FUNCTION_BLOCK FB_MapStim300
VAR_INPUT
	stFilterParams : ST_FTR_IIRSpec := (
		eFilterName   := E_FTR_Name.eButterworth,
		eFilterType   := E_FTR_Type.eLowPass,
		nFilterOrder  := 2,
		fSamplingRate := 0.001,
		fCutoff       := 4.0,
		nOversamples  := 1,
		nChannels     := 1,
		pInitialValues := ADR(fRollDeg),
		nInitialValuesSize := SIZEOF(fRollDeg)
	);
	
	fbFilter : FB_FTR_IIRSpec := (stConfig := stFilterParams);
END_VAR
VAR_OUTPUT
	ImuData : ST_IMUData;
	
	fRollDegFiltered : LREAL;
	fRollDeg : LREAL;
	fPitchDeg : LREAL;
END_VAR

VAR
		

	//serial communication with el6022
	fbGetSerialData : FB_GetSerialData;	
	ImuRawDataFrame : tDataFrame;
	
	fbEL6022Ctrl       : SerialLineControl;
	bEL6022CtrlError   : BOOL;
   	eEL6022CtrlErrorID : ComError_t;
   
	(* I/O variables for a EL6022 terminal*)
	stIn_EL6022 AT %I*    : EL6inData22B; 		(* linked to the EL6022 in the TwinCAT System Manager *)
	stOut_EL6022 AT %Q*    : EL6outData22B;		(* linked to the EL6022 in the TwinCAT System Manager *)
	
	RxBufferEL : ComBuffer; (* Receive data buffer; used with all receive function blocks *)
	TxBufferEL : ComBuffer; (* Transmit data buffer; used with all receive function blocks *)

	

	fbTimer : TON := (PT := T#1S);
	nCounter : DINT;
	fSampleRate : LREAL;
	
	//COmplementary filter
	fbAccelerometer : FB_AccelerometerAngle;
	fbComplementaryFilterRoll : FB_ComplementaryFilter := (fFilterRatio:=0.98);
	fbComplementaryFilterPitch : FB_ComplementaryFilter := (fFilterRatio:=0.98);
	
	// Task cycle time monitoring
	bFirstRun : BOOL := TRUE;
	Ts : LREAL := 0.01;
	fbGetCurrentTaskIdx : GETCURTASKINDEX;
	bCycleTimeExceeded : BOOL;
	nCycleCount : UDINT;
	
END_VAR

VAR CONSTANT
	header : BYTE := 16#AF;
	nDataSize : UDINT := SIZEOF(tDataFrame);
	fRatioGyro : LREAL := 1.0/EXPT(2,14);
	fRatioAcc : LREAL := 1.0/EXPT(2,19);
END_VAR

IF bFirstRun THEN
	getSampleTIme();
	bFirstRun:= FALSE;
END_IF

fbEL6022Ctrl(
   Mode:= SERIALLINEMODE_EL6_22B, 
   pComIn:= ADR(stIn_EL6022), 
   pComOut:= ADR(stOut_EL6022), 
   SizeComIn:= SIZEOF(stIn_EL6022), 
   Error=> bEL6022CtrlError, 
   ErrorID=> eEL6022CtrlErrorID, 
   TxBuffer:= TxBufferEL, 
   RxBuffer:= RxBufferEL
);

nCounter := nCounter + 1;
fbTimer(IN := TRUE);
IF fbTimer.Q THEN
	fbTimer(IN := FALSE);
	fSampleRate := 1.0/TO_LREAL(nCounter);
	nCounter := 0;
END_IF

fbGetSerialData(
	pHeader := ADR(header),
	cbHeaderSize := 1,
	cbPacketSize := nDataSize,
	stRxBuffer := RxBufferEL,
	pDataBuffer := ADR(ImuRawDataFrame),
	cbDataBufferSize := nDataSize
);

IF fbGetSerialData.NewData THEN
	mapStim300(
		in := ADR(ImuRawDataFrame),
		out := ImuData
	);
	
	fbAccelerometer(fAx:=ImuData.stAcc.x,fAy:=ImuData.stAcc.y,fAz:=ImuData.stAcc.z);
	
	
END_IF

fbComplementaryFilterRoll(fAccAngle:=fbAccelerometer.fRoll,fGyroRate:=ImuData.stGyro.x*CONSTANTS.DEG_TO_RAD,fStepTime:=Ts,fAngle=>ImuData.fRoll);
fbComplementaryFilterPitch(fAccAngle:=fbAccelerometer.fPitch,fGyroRate:=ImuData.stGyro.y*CONSTANTS.DEG_TO_RAD,fStepTime:=Ts,fAngle=>ImuData.fPitch);

fRollDeg := ImuData.fRoll * CONSTANTS.RAD_TO_DEG;
fbFilter.Call(
	pIn := ADR(fRollDeg),
	nSizeIn := SIZEOF(fRollDeg),
	pOut := ADR(fRollDegFiltered),
	nSizeOut := SIZEOF(fRollDegFiltered)
);

fPitchDeg := ImuData.fPitch * CONSTANTS.RAD_TO_DEG;

ACTION getSampleTIme:
// Get sample time of current task
fbGetCurrentTaskIdx();
bCycleTimeExceeded := _TaskInfo[fbGetCurrentTaskIdx.index].CycleTimeExceeded;
nCycleCount := _TaskInfo[fbGetCurrentTaskIdx.index].CycleCount;
Ts := UDINT_TO_LREAL(_TaskInfo[fbGetCurrentTaskIdx.index].CycleTime/10)/1E6;
//stFilterParams.fSamplingRate := Ts;
END_ACTION

METHOD PUBLIC mapStim300
VAR_INPUT
	in 	: POINTER TO BYTE;
	out : REFERENCE TO ST_ImuData;
END_VAR
	
	out.stGyro.x := TO_LREAL(F_Merge24BitSigned(in[1], in[2], in[3]))*fRatioGyro;
	out.stGyro.y := TO_LREAL(F_Merge24BitSigned(in[4], in[5], in[6]))*fRatioGyro;
	out.stGyro.z := TO_LREAL(F_Merge24BitSigned(in[7], in[8], in[9]))*fRatioGyro;
	
	out.stAcc.x := TO_LREAL(F_Merge24BitSigned(in[11], in[12], in[13]))*fRatioAcc;
	out.stAcc.y := TO_LREAL(F_Merge24BitSigned(in[14], in[15], in[16]))*fRatioAcc;
	out.stAcc.z := TO_LREAL(F_Merge24BitSigned(in[17], in[18], in[19]))*fRatioAcc;
END_METHOD

END_FUNCTION_BLOCK

(* stored: Version 1.1.0.1, ProductVersion 3.1.4024.3
   POU FB_MapStim300: Id {5f7fd0be-53b8-4cf8-b0c9-21f376e0f253}, SpecialFunc None
   Action getSampleTIme: Id {cb4477fb-985f-4474-b442-53511ea0cc37}
   Method mapStim300: Id {cbc54e7b-fbd0-4f47-86b5-0d52db7252fa} *)
